PROGRAM P_6Stack
VAR
	nState: INT;
	
	//Timers
	fbTimerMovingLoad: TON;
	fbTimerLift: TON;
	fbTimerToSpace: TON;
	fbTimerPlace: TON;
	fbTimerCounter: TON;
	fbTimerHoming: TON;
	
	
	AtLoadTrig:R_TRIG;		

	//INT
	nCounter         : INT := 0;
END_VAR

VAR CONSTANT
	//Here we define our constant where we want the different positon to be. This is instead of making steps you can call this fixed steps.
	Start		:INT:=00;
	AtLoad		:INT:=01;
	PickUP 		:INT := 02;
	LiftPallet         : INT := 03;
	RetractForksLeft   : INT := 04;
	MovingToSpace      : INT := 05;
	DeliverPart        : INT := 06;
	PlacePallet        : INT := 07;
	RetractRight       : INT := 08;
	Homing             : INT := 09;
	Retry   		   : INT := 10;
	Moving     : INT := 20;
	MovingStop : INT := 22;
	GetPart            : INT := 50;
	GetPartPick        : INT := 51;
	PartPickUp    	   : INT := 52;
	PickUpPart         : INT := 53;
	PartPicked 		   : INT := 54;
	MoveToUnload       : INT := 55;
	UnloadPart 		   : INT := 56;
	PlacePart          : INT := 57;
	Waiting    : INT := 30;	
	Stopping   : INT := 40;
	Resetting  : INT := 60;
	Estop      : INT := 9999;		
END_VAR

// This is our sixth program the stacker robot will pick up the pallet at load and stack them into the different shelf from 1 to 54. 


AtLoadTrig(CLK:=FIO.bScAtLoad);


CASE nState OF
		Start: //Entry of the Palled 
			IF FIO.bScAtLoad=FALSE AND FIO.bScConv3=TRUE THEN
				FIO.bScLoadingConv:=TRUE;                       //turning on the load conveyor
			END_IF
				FIO.iSC_TargetPos := 21474; //This is the value that sends the crane home.
			
			IF AtLoadTrig.Q THEN // counter for the stack robot to know which shelf to put the palled in shelf no = anount of pallet that have been at entry.
			nCounter:=nCounter+1;
			END_IF
			IF FIO.bScAtLoad=TRUE THEN
				nState := AtLoad;
			END_IF
		
		AtLoad:	 // Pallet is at load, the different conveyor will go false when pallet is at load.
		IF FIO.bScAtLoad=TRUE THEN 
			FIO.bScLoadingConv:=FALSE;
			fbTimerMovingLoad(IN:=TRUE,PT:=T#1S);
			IF fbTimerMovingLoad.Q THEN
				fbTimerMovingLoad(IN:=FALSE);
				FIO.bScConv3:=FALSE;
				nState := PickUP;
		 	END_IF						
		END_IF	

	PickUP:  // here we make sure that the the stack robot are at home and there pallet at the load and moving x and z are false before it cna pick up a pallet.
		IF FIO.bScAtLoad=TRUE AND FIO.iSC_TargetPos = 21474 AND FIO.bSC_MovingX=FALSE and FIO.bSC_MovingZ=FALSE THEN
			FIO.bSc_Left := TRUE;
			nState := LiftPallet;
		END_IF
	
	LiftPallet:	 // there the pallet gets picked up	
		IF FIO.bSc_AtLeft=TRUE THEN
			FIO.bSc_Lift:=TRUE;
			fbTimerLift(IN:=TRUE,PT:=T#1S);	
			IF fbTimerLift.Q THEN
				fbTimerLift(IN:=FALSE);
				FIO.bSc_Left :=FALSE; 
				nState := RetractForksLeft;
			END_IF	
		END_IF
	
	RetractForksLeft:  // here er made an extra step to give time for the fock to come back before we move to the next state
			nState:= MovingToSpace;
			
	MovingToSpace:	// here we make sure that the pallet are at mid before the stack robot moves again and we cound which palle 
		IF 	FIO.bSC_AtMiddle=TRUE THEN
			FIO.iSC_TargetPos:=nCounter;    //here we set the pallet count = the target pos which is the space in the shelf
			fbTimerToSpace(IN:=TRUE,PT:=T#2S);	
			IF fbTimerToSpace.Q THEN
				fbTimerToSpace(IN:=FALSE);
				nState := DeliverPart;
			END_IF
		END_IF

	DeliverPart: // here we put pallet into shelf                             
		IF FIO.bSC_MovingX=FALSE THEN
		FIO.bSc_Right := TRUE;                    
		nState := PlacePallet;
		END_IF
		
	PlacePallet:   
		IF FIO.bSc_AtRight=TRUE THEN
			FIO.bSc_Lift:=FALSE;
			fbTimerPlace(IN:=TRUE,PT:=T#1S);	
			IF fbTimerPlace.Q THEN
				fbTimerPlace(IN:=FALSE);
				nState := RetractRight;
			END_IF	
		END_IF

   		RetractRight:   //retract the arm     
		    IF FIO.bSc_Lift=FALSE THEN
				FIO.bSc_Right:=FALSE;
			fbTimerHoming(IN:=TRUE,PT:=T#1S);	
			IF fbTimerHoming.Q THEN
				fbTimerHoming(IN:=FALSE);
				nState := Homing; 		
			END_IF				
		END_IF

	Homing:		//moving to homing
		IF FIO.bSc_AtMiddle=TRUE THEN
			FIO.iSc_TargetPos := 21474;
			nState := Start;	
		END_IF		
		
	ELSE

	nState:=9999;		
	
END_CASE

END_PROGRAM

(* stored: Version 1.1.0.1, ProductVersion 3.1.4024.3
   POU P_6Stack: Id {20ac5aef-e629-4ad3-b29a-76974f20f0ec}, SpecialFunc None *)
